FUNCTION_BLOCK F_CONCAT_DATE_TOD (* concatenation *)
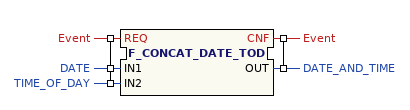
  EVENT_INPUT
    REQ WITH IN1, IN2; (* Service Request *)
  END_EVENT
  EVENT_OUTPUT
    CNF WITH OUT; (* Confirmation of Requested Service *)
  END_EVENT
  VAR_INPUT
    IN1 : DATE; (* date input *)
    IN2 : TIME_OF_DAY; (* time of day input *)
  END_VAR
  VAR_OUTPUT
    OUT : DATE_AND_TIME; (* date + time of day *)
  END_VAR
END_FUNCTION_BLOCK
